TYPE T_COMMHANDLE : ARRAY[0..24] OF USINT; END_TYPE

(* stored: Version 1.1.0.1, ProductVersion 3.1.4019.2
   DUT T_COMMHANDLE: Id {c2b205fa-0a9f-4377-bcb0-6a7577aabc59} *)
